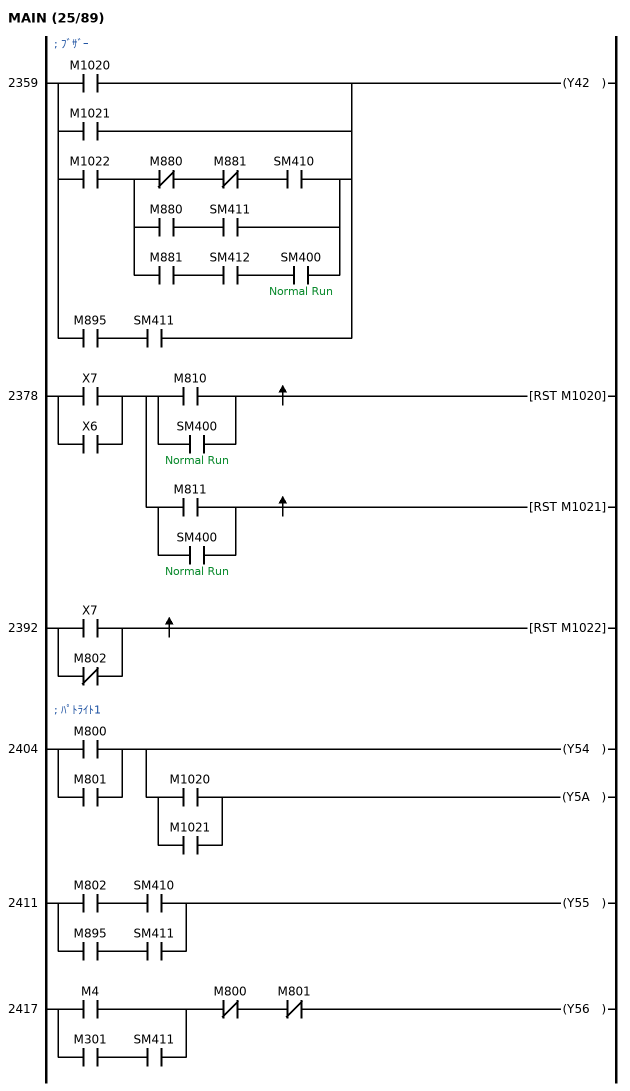
[picture p24: ladder of MAIN, rungs at steps 2359 to 2417]
; ﾌﾞｻﾞｰ
2359  LD      M1020
      OR      M1021
      LD      M1022
      LDI     M880
      ANI     M881
      AND     SM410
      LD      M880
      AND     SM411
      ORB
      LD      M881
      AND     SM412
      AND     SM400  ; Normal Run
      ORB
      ANB
      ORB
      LD      M895
      AND     SM411
      ORB
      OUT     Y42
2378  LD      X7
      OR      X6
      MPS
      LD      M810
      OR      SM400  ; Normal Run
      ANB
      MEP
      RST     M1020
      MPP
      LD      M811
      OR      SM400  ; Normal Run
      ANB
      MEP
      RST     M1021
2392  LD      X7
      ORI     M802
      MEP
      RST     M1022
; ﾊﾟﾄﾗｲﾄ1
2404  LD      M800
      OR      M801
      OUT     Y54
      LD      M1020
      OR      M1021
      ANB
      OUT     Y5A
2411  LD      M802
      AND     SM410
      LD      M895
      AND     SM411
      ORB
      OUT     Y55
2417  LD      M4
      LD      M301
      AND     SM411
      ORB
      ANI     M800
      ANI     M801
      OUT     Y56
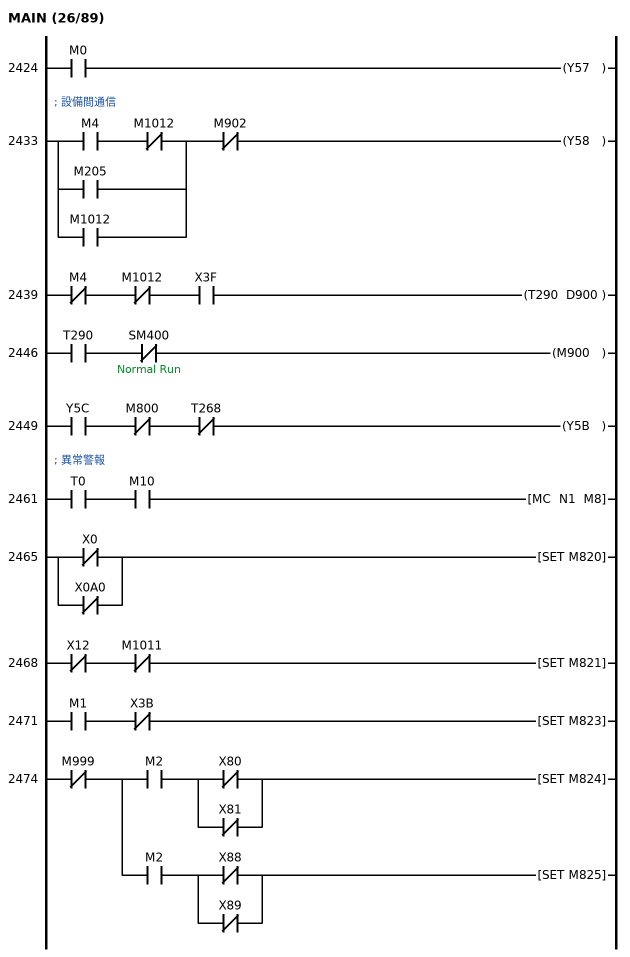
2424  LD      M0
      OUT     Y57
; 設備間通信
2433  LD      M4
      ANI     M1012
      OR      M205
      OR      M1012
      ANI     M902
      OUT     Y58
2439  LDI     M4
      ANI     M1012
      AND     X3F
      OUT     T290 D900
2446  LD      T290
      ANI     SM400  ; Normal Run
      OUT     M900
2449  LD      Y5C
      ANI     M800
      ANI     T268
      OUT     Y5B
; 異常警報
; 
2461  LD      T0
      AND     M10
      MC      N1 M8
2465  LDI     X0
      ORI     X0A0
      SET     M820
2468  LDI     X12
      ANI     M1011
      SET     M821
2471  LD      M1
      ANI     X3B
      SET     M823
2474  LDI     M999
      MPS
      AND     M2
      LDI     X80
      ORI     X81
      ANB
      SET     M824
      MPP
      AND     M2
      LDI     X88
      ORI     X89
      ANB
      SET     M825
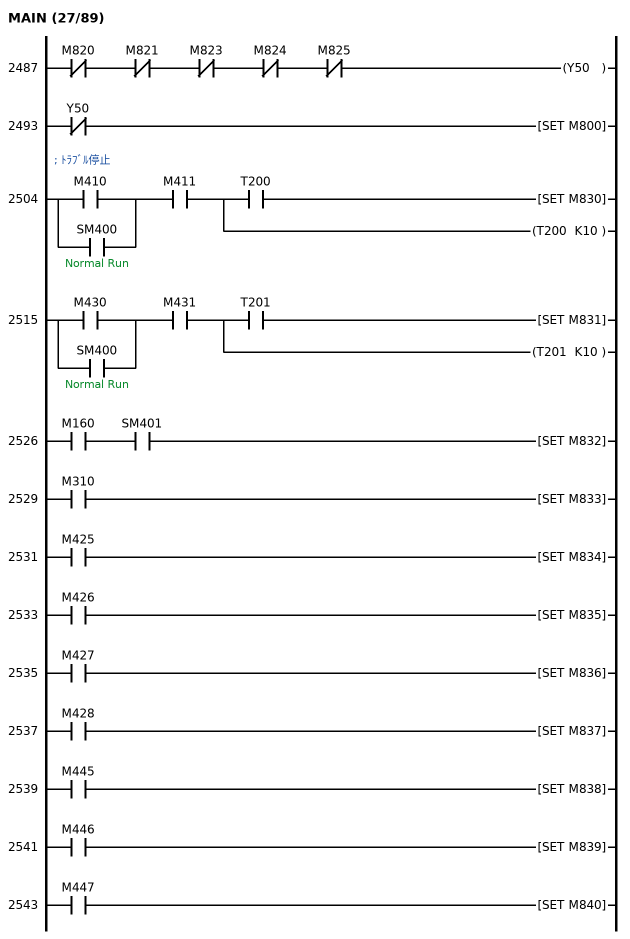
2487  LDI     M820
      ANI     M821
      ANI     M823
      ANI     M824
      ANI     M825
      OUT     Y50
2493  LDI     Y50
      SET     M800
; ﾄﾗﾌﾞﾙ停止
2504  LD      M410
      OR      SM400  ; Normal Run
      AND     M411
      MPS
      AND     T200
      SET     M830
      MPP
      OUT     T200 K10
2515  LD      M430
      OR      SM400  ; Normal Run
      AND     M431
      MPS
      AND     T201
      SET     M831
      MPP
      OUT     T201 K10
2526  LD      M160
      AND     SM401
      SET     M832
2529  LD      M310
      SET     M833
2531  LD      M425
      SET     M834
2533  LD      M426
      SET     M835
2535  LD      M427
      SET     M836
2537  LD      M428
      SET     M837
2539  LD      M445
      SET     M838
2541  LD      M446
      SET     M839
2543  LD      M447
      SET     M840
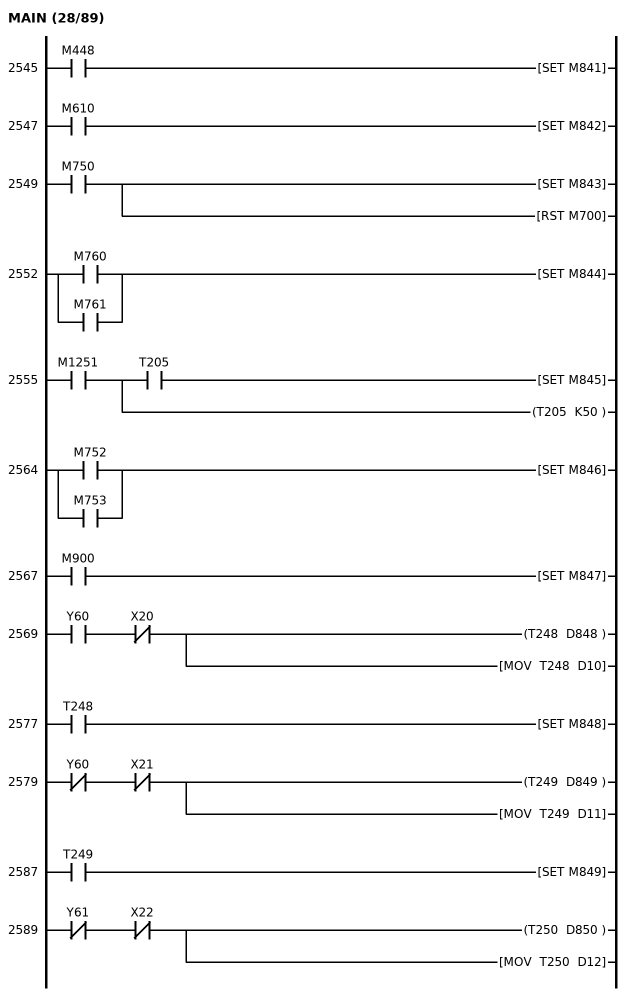
2545  LD      M448
      SET     M841
2547  LD      M610
      SET     M842
2549  LD      M750
      SET     M843
      RST     M700
2552  LD      M760
      OR      M761
      SET     M844
2555  LD      M1251
      MPS
      AND     T205
      SET     M845
      MPP
      OUT     T205 K50
2564  LD      M752
      OR      M753
      SET     M846
2567  LD      M900
      SET     M847
2569  LD      Y60
      ANI     X20
      OUT     T248 D848
      MOV     T248 D10
2577  LD      T248
      SET     M848
2579  LDI     Y60
      ANI     X21
      OUT     T249 D849
      MOV     T249 D11
2587  LD      T249
      SET     M849
2589  LDI     Y61
      ANI     X22
      OUT     T250 D850
      MOV     T250 D12
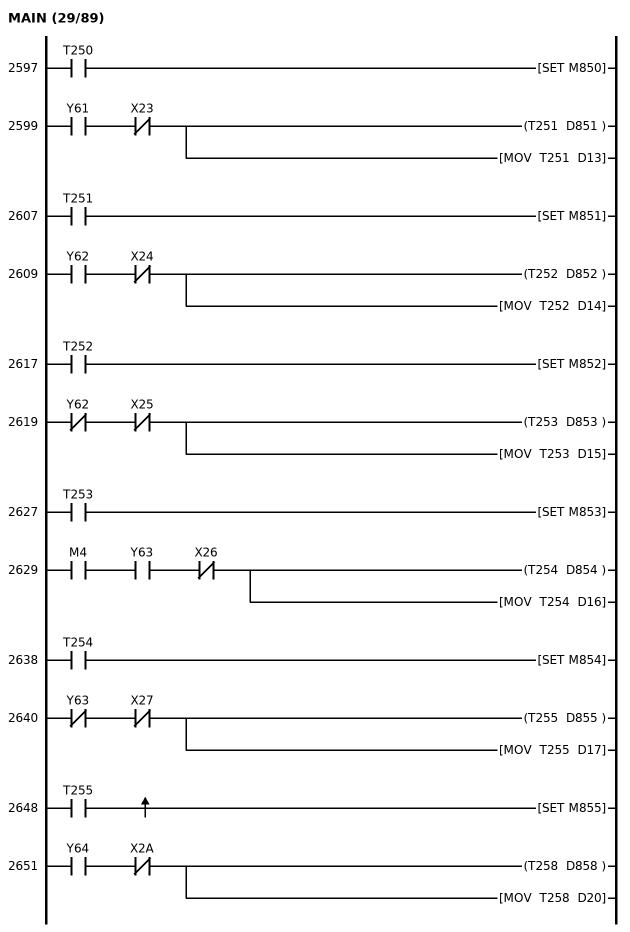
2597  LD      T250
      SET     M850
2599  LD      Y61
      ANI     X23
      OUT     T251 D851
      MOV     T251 D13
2607  LD      T251
      SET     M851
2609  LD      Y62
      ANI     X24
      OUT     T252 D852
      MOV     T252 D14
2617  LD      T252
      SET     M852
2619  LDI     Y62
      ANI     X25
      OUT     T253 D853
      MOV     T253 D15
2627  LD      T253
      SET     M853
2629  LD      M4
      AND     Y63
      ANI     X26
      OUT     T254 D854
      MOV     T254 D16
2638  LD      T254
      SET     M854
2640  LDI     Y63
      ANI     X27
      OUT     T255 D855
      MOV     T255 D17
2648  LD      T255
      MEP
      SET     M855
2651  LD      Y64
      ANI     X2A
      OUT     T258 D858
      MOV     T258 D20
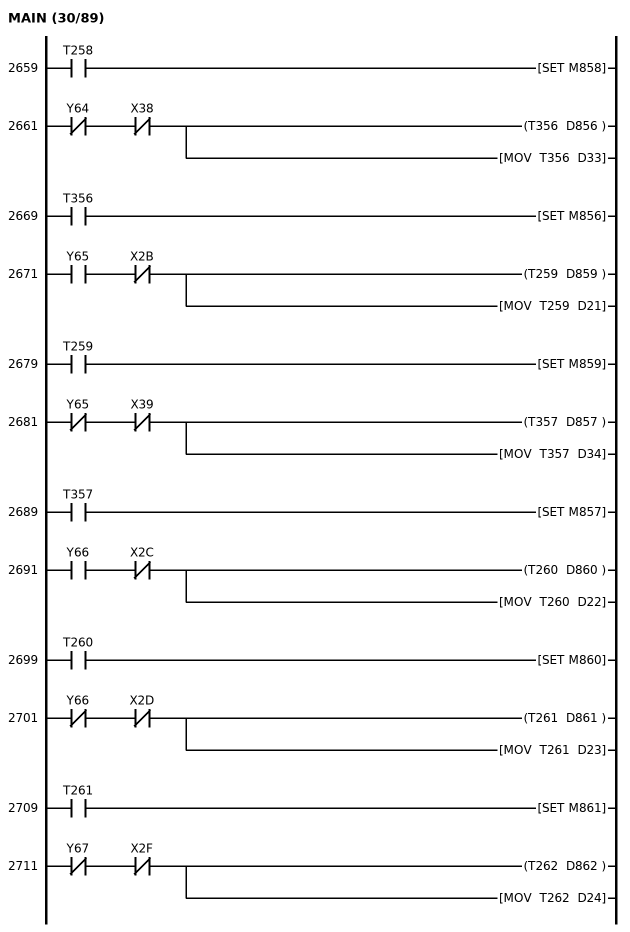
2659  LD      T258
      SET     M858
2661  LDI     Y64
      ANI     X38
      OUT     T356 D856
      MOV     T356 D33
2669  LD      T356
      SET     M856
2671  LD      Y65
      ANI     X2B
      OUT     T259 D859
      MOV     T259 D21
2679  LD      T259
      SET     M859
2681  LDI     Y65
      ANI     X39
      OUT     T357 D857
      MOV     T357 D34
2689  LD      T357
      SET     M857
2691  LD      Y66
      ANI     X2C
      OUT     T260 D860
      MOV     T260 D22
2699  LD      T260
      SET     M860
2701  LDI     Y66
      ANI     X2D
      OUT     T261 D861
      MOV     T261 D23
2709  LD      T261
      SET     M861
2711  LDI     Y67
      ANI     X2F
      OUT     T262 D862
      MOV     T262 D24
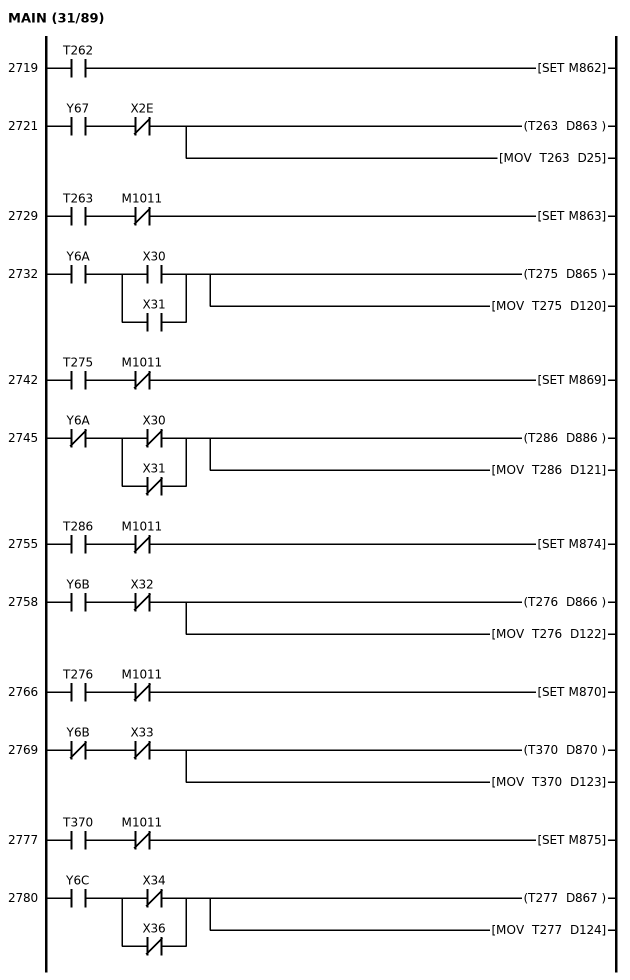
2719  LD      T262
      SET     M862
2721  LD      Y67
      ANI     X2E
      OUT     T263 D863
      MOV     T263 D25
2729  LD      T263
      ANI     M1011
      SET     M863
2732  LD      Y6A
      LD      X30
      OR      X31
      ANB
      OUT     T275 D865
      MOV     T275 D120
2742  LD      T275
      ANI     M1011
      SET     M869
2745  LDI     Y6A
      LDI     X30
      ORI     X31
      ANB
      OUT     T286 D886
      MOV     T286 D121
2755  LD      T286
      ANI     M1011
      SET     M874
2758  LD      Y6B
      ANI     X32
      OUT     T276 D866
      MOV     T276 D122
2766  LD      T276
      ANI     M1011
      SET     M870
2769  LDI     Y6B
      ANI     X33
      OUT     T370 D870
      MOV     T370 D123
2777  LD      T370
      ANI     M1011
      SET     M875
2780  LD      Y6C
      LDI     X34
      ORI     X36
      ANB
      OUT     T277 D867
      MOV     T277 D124
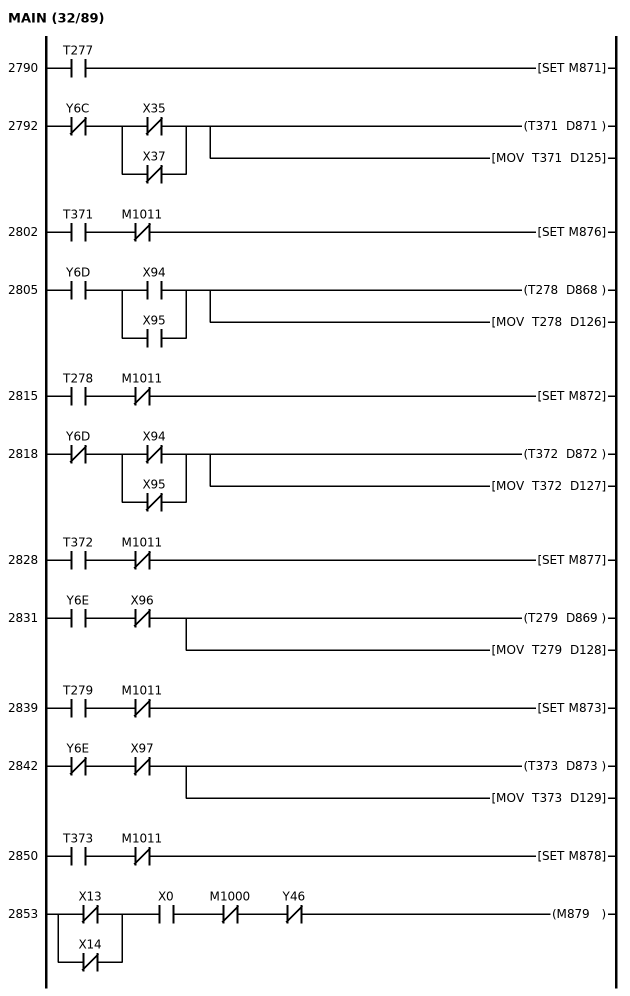
2790  LD      T277
      SET     M871
2792  LDI     Y6C
      LDI     X35
      ORI     X37
      ANB
      OUT     T371 D871
      MOV     T371 D125
2802  LD      T371
      ANI     M1011
      SET     M876
2805  LD      Y6D
      LD      X94
      OR      X95
      ANB
      OUT     T278 D868
      MOV     T278 D126
2815  LD      T278
      ANI     M1011
      SET     M872
2818  LDI     Y6D
      LDI     X94
      ORI     X95
      ANB
      OUT     T372 D872
      MOV     T372 D127
2828  LD      T372
      ANI     M1011
      SET     M877
2831  LD      Y6E
      ANI     X96
      OUT     T279 D869
      MOV     T279 D128
2839  LD      T279
      ANI     M1011
      SET     M873
2842  LDI     Y6E
      ANI     X97
      OUT     T373 D873
      MOV     T373 D129
2850  LD      T373
      ANI     M1011
      SET     M878
2853  LDI     X13
      ORI     X14
      AND     X0
      ANI     M1000
      ANI     Y46
      OUT     M879
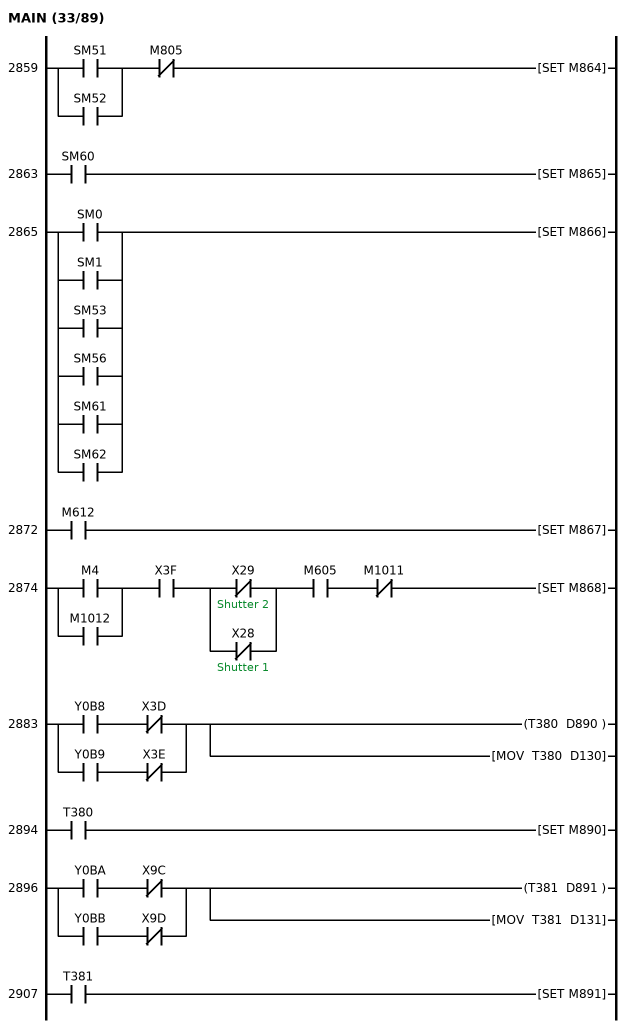
2859  LD      SM51
      OR      SM52
      ANI     M805
      SET     M864
2863  LD      SM60
      SET     M865
2865  LD      SM0
      OR      SM1
      OR      SM53
      OR      SM56
      OR      SM61
      OR      SM62
      SET     M866
2872  LD      M612
      SET     M867
2874  LD      M4
      OR      M1012
      AND     X3F
      LDI     X29  ; Shutter 2
      ORI     X28  ; Shutter 1
      ANB
      AND     M605
      ANI     M1011
      SET     M868
2883  LD      Y0B8
      ANI     X3D
      LD      Y0B9
      ANI     X3E
      ORB
      OUT     T380 D890
      MOV     T380 D130
2894  LD      T380
      SET     M890
2896  LD      Y0BA
      ANI     X9C
      LD      Y0BB
      ANI     X9D
      ORB
      OUT     T381 D891
      MOV     T381 D131
2907  LD      T381
      SET     M891
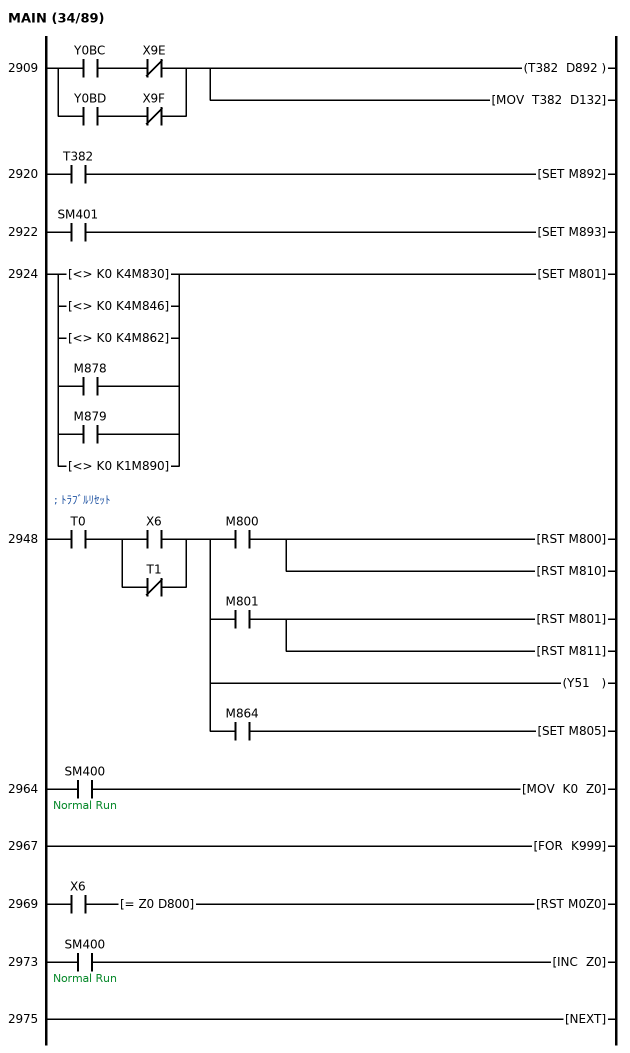
2909  LD      Y0BC
      ANI     X9E
      LD      Y0BD
      ANI     X9F
      ORB
      OUT     T382 D892
      MOV     T382 D132
2920  LD      T382
      SET     M892
2922  LD      SM401
      SET     M893
2924  LD<>    K0 K4M830
      OR<>    K0 K4M846
      OR<>    K0 K4M862
      OR      M878
      OR      M879
      OR<>    K0 K1M890
      SET     M801
; ﾄﾗﾌﾞﾙﾘｾｯﾄ
2948  LD      T0
      LD      X6
      ORI     T1
      ANB
      MPS
      AND     M800
      RST     M800
      RST     M810
      MRD
      AND     M801
      RST     M801
      RST     M811
      MPP
      OUT     Y51
      AND     M864
      SET     M805
2964  LD      SM400  ; Normal Run
      MOV     K0 Z0
2967  FOR     K999
2969  LD      X6
      AND=    Z0 D800
      RST     M0Z0
2973  LD      SM400  ; Normal Run
      INC     Z0
2975  NEXT
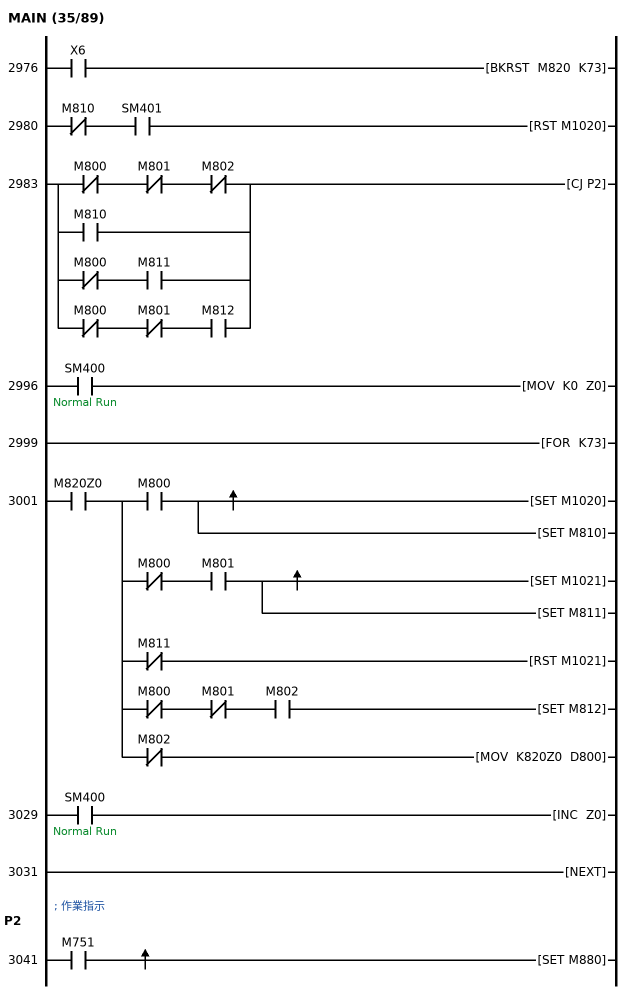
2976  LD      X6
      BKRST   M820 K73
2980  LDI     M810
      AND     SM401
      RST     M1020
2983  LDI     M800
      ANI     M801
      ANI     M802
      OR      M810
      LDI     M800
      AND     M811
      ORB
      LDI     M800
      ANI     M801
      AND     M812
      ORB
      CJ      P2
2996  LD      SM400  ; Normal Run
      MOV     K0 Z0
2999  FOR     K73
3001  LD      M820Z0
      MPS
      AND     M800
      MPS
      MEP
      SET     M1020
      MPP
      SET     M810
      MRD
      ANI     M800
      AND     M801
      MPS
      MEP
      SET     M1021
      MPP
      SET     M811
      MRD
      ANI     M811
      RST     M1021
      MRD
      ANI     M800
      ANI     M801
      AND     M802
      SET     M812
      MPP
      ANI     M802
      MOV     K820Z0 D800
3029  LD      SM400  ; Normal Run
      INC     Z0
3031  NEXT
      P2
; 作業指示
3041  LD      M751
      MEP
      SET     M880
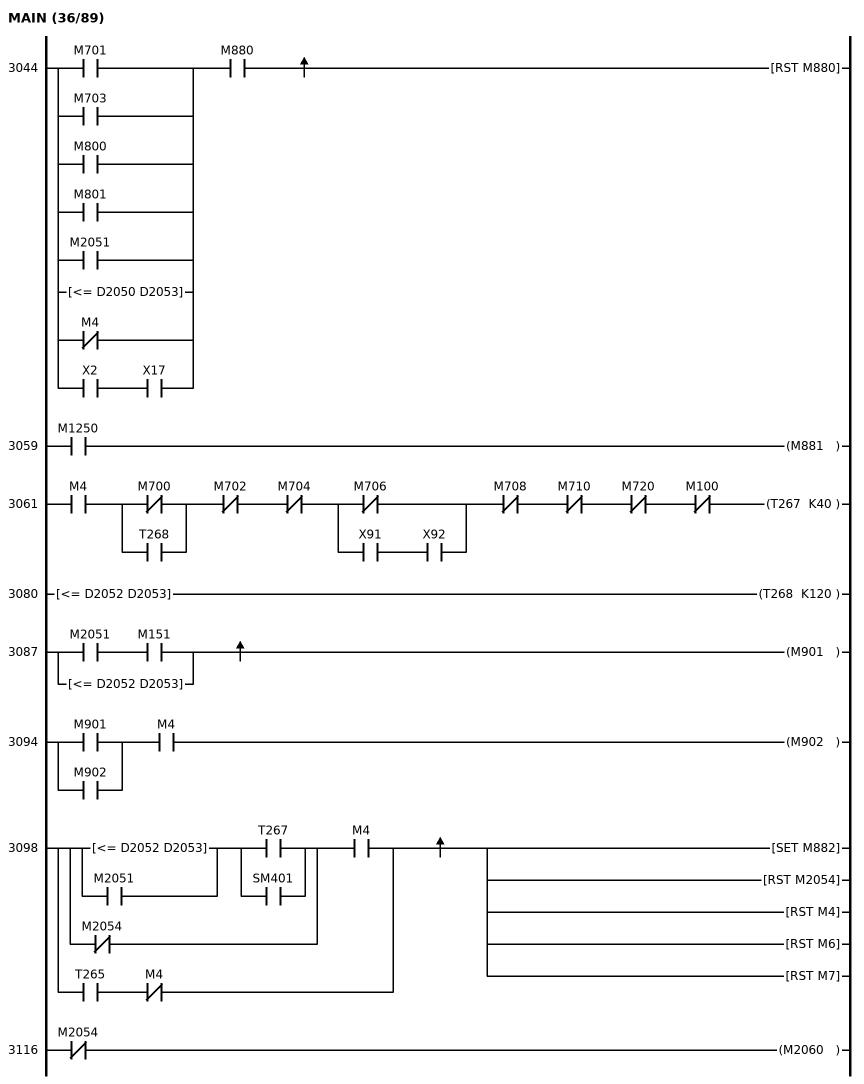
3044  LD      M701
      OR      M703
      OR      M800
      OR      M801
      OR      M2051
      OR<=    D2050 D2053
      ORI     M4
      LD      X2
      AND     X17
      ORB
      AND     M880
      MEP
      RST     M880
3059  LD      M1250
      OUT     M881
3061  LD      M4
      LDI     M700
      OR      T268
      ANB
      ANI     M702
      ANI     M704
      LDI     M706
      LD      X91
      AND     X92
      ORB
      ANB
      ANI     M708
      ANI     M710
      ANI     M720
      ANI     M100
      OUT     T267 K40
3080  LD<=    D2052 D2053
      OUT     T268 K120
3087  LD      M2051
      AND     M151
      OR<=    D2052 D2053
      MEP
      OUT     M901
3094  LD      M901
      OR      M902
      AND     M4
      OUT     M902
3098  LD<=    D2052 D2053
      OR      M2051
      LD      T267
      OR      SM401
      ANB
      ORI     M2054
      AND     M4
      LD      T265
      ANI     M4
      ORB
      MEP
      SET     M882
      RST     M2054
      RST     M4
      RST     M6
      RST     M7
3116  LDI     M2054
      OUT     M2060
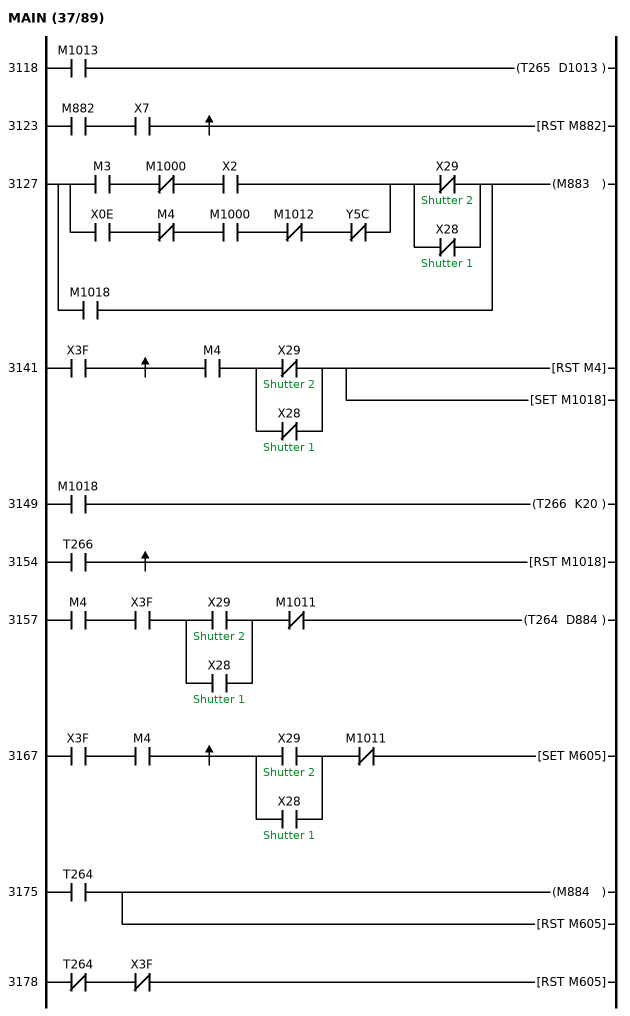
3118  LD      M1013
      OUT     T265 D1013
3123  LD      M882
      AND     X7
      MEP
      RST     M882
3127  LD      M3
      ANI     M1000
      AND     X2
      LD      X0E
      ANI     M4
      AND     M1000
      ANI     M1012
      ANI     Y5C
      ORB
      LDI     X29  ; Shutter 2
      ORI     X28  ; Shutter 1
      ANB
      OR      M1018
      OUT     M883
3141  LD      X3F
      MEP
      AND     M4
      LDI     X29  ; Shutter 2
      ORI     X28  ; Shutter 1
      ANB
      RST     M4
      SET     M1018
3149  LD      M1018
      OUT     T266 K20
3154  LD      T266
      MEP
      RST     M1018
3157  LD      M4
      AND     X3F
      LD      X29  ; Shutter 2
      OR      X28  ; Shutter 1
      ANB
      ANI     M1011
      OUT     T264 D884
3167  LD      X3F
      AND     M4
      MEP
      LD      X29  ; Shutter 2
      OR      X28  ; Shutter 1
      ANB
      ANI     M1011
      SET     M605
3175  LD      T264
      OUT     M884
      RST     M605
3178  LDI     T264
      ANI     X3F
      RST     M605
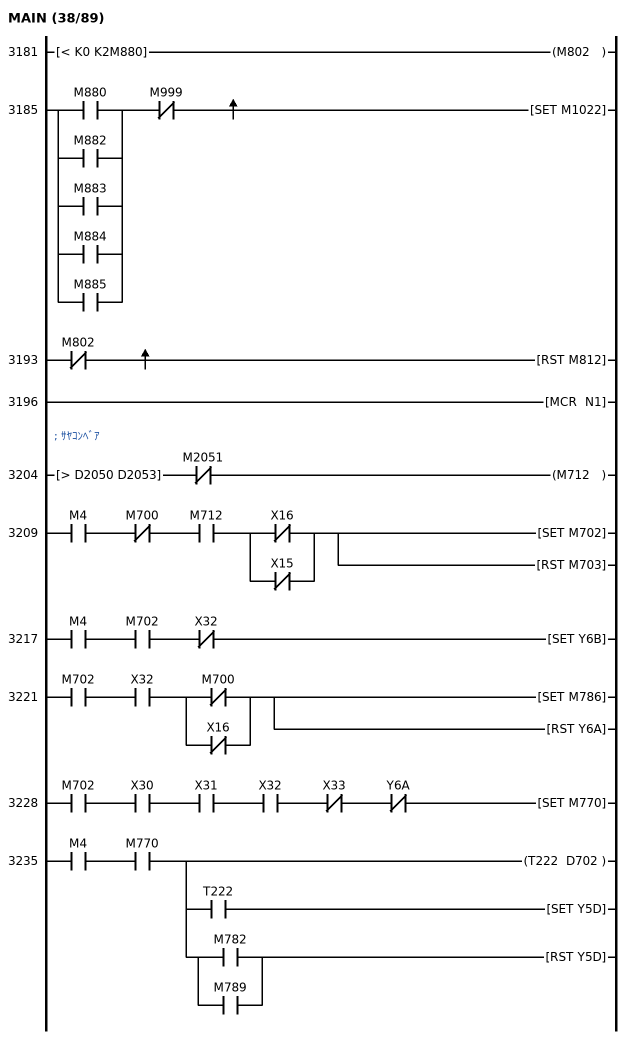
3181  LD<     K0 K2M880
      OUT     M802
3185  LD      M880
      OR      M882
      OR      M883
      OR      M884
      OR      M885
      ANI     M999
      MEP
      SET     M1022
3193  LDI     M802
      MEP
      RST     M812
3196  MCR     N1
; ｻﾔｺﾝﾍﾞｱ
; 
3204  LD>     D2050 D2053
      ANI     M2051
      OUT     M712
3209  LD      M4
      ANI     M700
      AND     M712
      LDI     X16
      ORI     X15
      ANB
      SET     M702
      RST     M703
3217  LD      M4
      AND     M702
      ANI     X32
      SET     Y6B
3221  LD      M702
      AND     X32
      LDI     M700
      ORI     X16
      ANB
      SET     M786
      RST     Y6A
3228  LD      M702
      AND     X30
      AND     X31
      AND     X32
      ANI     X33
      ANI     Y6A
      SET     M770
3235  LD      M4
      AND     M770
      OUT     T222 D702
      MPS
      AND     T222
      SET     Y5D
      MPP
      LD      M782
      OR      M789
      ANB
      RST     Y5D
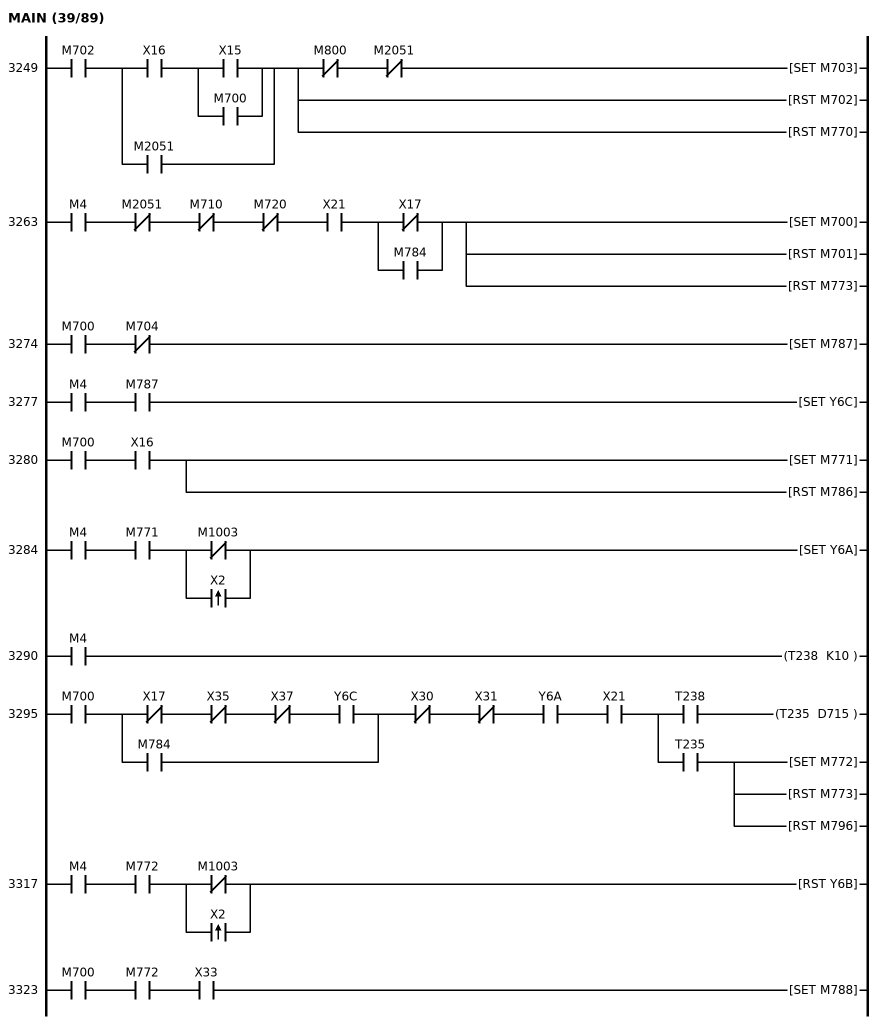
3249  LD      M702
      LD      X16
      LD      X15
      OR      M700
      ANB
      OR      M2051
      ANB
      MPS
      ANI     M800
      ANI     M2051
      SET     M703
      MPP
      RST     M702
      RST     M770
3263  LD      M4
      ANI     M2051
      ANI     M710
      ANI     M720
      AND     X21
      LDI     X17
      OR      M784
      ANB
      SET     M700
      RST     M701
      RST     M773
3274  LD      M700
      ANI     M704
      SET     M787
3277  LD      M4
      AND     M787
      SET     Y6C
3280  LD      M700
      AND     X16
      SET     M771
      RST     M786
3284  LD      M4
      AND     M771
      LDI     M1003
      ORP     X2
      ANB
      SET     Y6A
3290  LD      M4
      OUT     T238 K10
3295  LD      M700
      LDI     X17
      ANI     X35
      ANI     X37
      AND     Y6C
      OR      M784
      ANB
      ANI     X30
      ANI     X31
      AND     Y6A
      AND     X21
      MPS
      AND     T238
      OUT     T235 D715
      MPP
      AND     T235
      SET     M772
      RST     M773
      RST     M796
3317  LD      M4
      AND     M772
      LDI     M1003
      ORP     X2
      ANB
      RST     Y6B
3323  LD      M700
      AND     M772
      AND     X33
      SET     M788
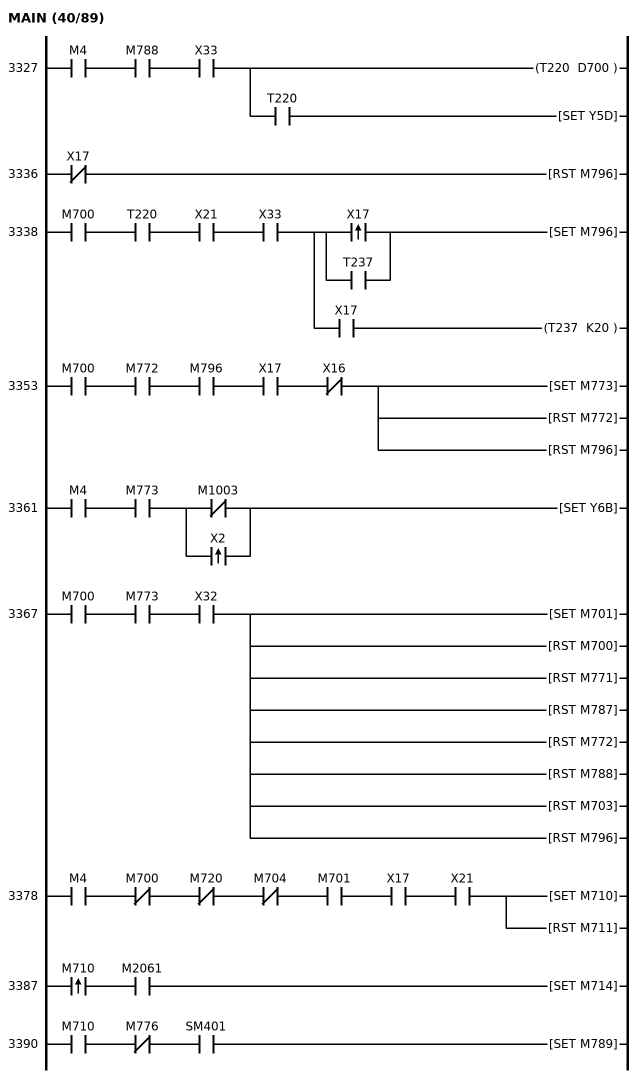
3327  LD      M4
      AND     M788
      AND     X33
      OUT     T220 D700
      AND     T220
      SET     Y5D
3336  LDI     X17
      RST     M796
3338  LD      M700
      AND     T220
      AND     X21
      AND     X33
      MPS
      LDP     X17
      OR      T237
      ANB
      SET     M796
      MPP
      AND     X17
      OUT     T237 K20
3353  LD      M700
      AND     M772
      AND     M796
      AND     X17
      ANI     X16
      SET     M773
      RST     M772
      RST     M796
3361  LD      M4
      AND     M773
      LDI     M1003
      ORP     X2
      ANB
      SET     Y6B
3367  LD      M700
      AND     M773
      AND     X32
      SET     M701
      RST     M700
      RST     M771
      RST     M787
      RST     M772
      RST     M788
      RST     M703
      RST     M796
3378  LD      M4
      ANI     M700
      ANI     M720
      ANI     M704
      AND     M701
      AND     X17
      AND     X21
      SET     M710
      RST     M711
3387  LDP     M710
      AND     M2061
      SET     M714
3390  LD      M710
      ANI     M776
      AND     SM401
      SET     M789
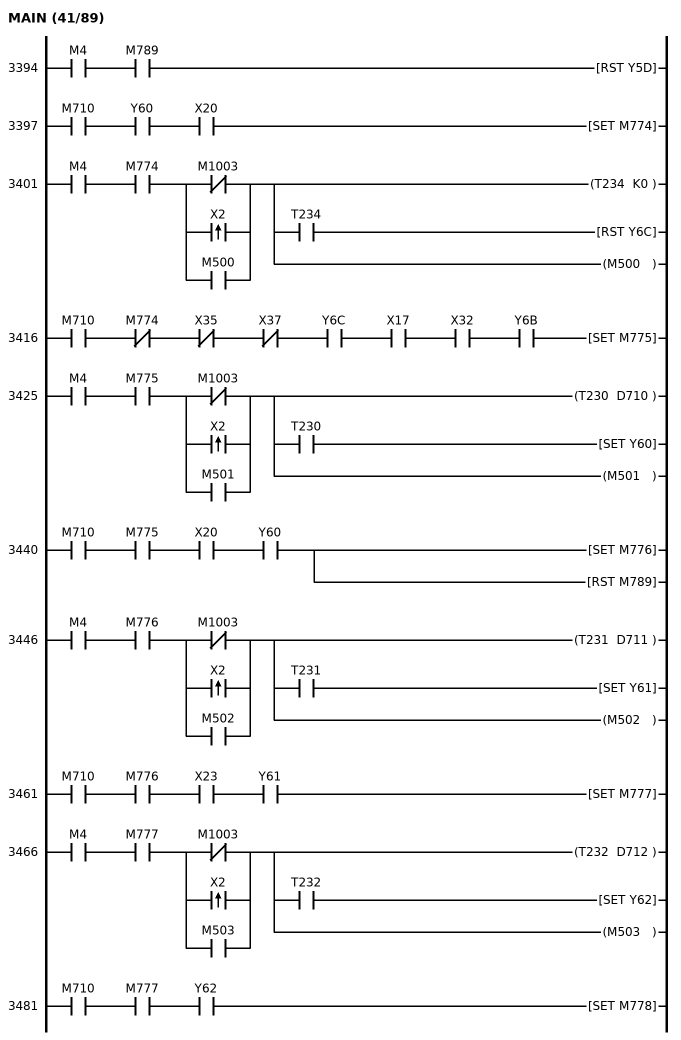
3394  LD      M4
      AND     M789
      RST     Y5D
3397  LD      M710
      AND     Y60
      AND     X20
      SET     M774
3401  LD      M4
      AND     M774
      LDI     M1003
      ORP     X2
      OR      M500
      ANB
      OUT     T234 K0
      MPS
      AND     T234
      RST     Y6C
      MPP
      OUT     M500
3416  LD      M710
      ANI     M774
      ANI     X35
      ANI     X37
      AND     Y6C
      AND     X17
      AND     X32
      AND     Y6B
      SET     M775
3425  LD      M4
      AND     M775
      LDI     M1003
      ORP     X2
      OR      M501
      ANB
      OUT     T230 D710
      MPS
      AND     T230
      SET     Y60
      MPP
      OUT     M501
3440  LD      M710
      AND     M775
      AND     X20
      AND     Y60
      SET     M776
      RST     M789
3446  LD      M4
      AND     M776
      LDI     M1003
      ORP     X2
      OR      M502
      ANB
      OUT     T231 D711
      MPS
      AND     T231
      SET     Y61
      MPP
      OUT     M502
3461  LD      M710
      AND     M776
      AND     X23
      AND     Y61
      SET     M777
3466  LD      M4
      AND     M777
      LDI     M1003
      ORP     X2
      OR      M503
      ANB
      OUT     T232 D712
      MPS
      AND     T232
      SET     Y62
      MPP
      OUT     M503
3481  LD      M710
      AND     M777
      AND     Y62
      SET     M778
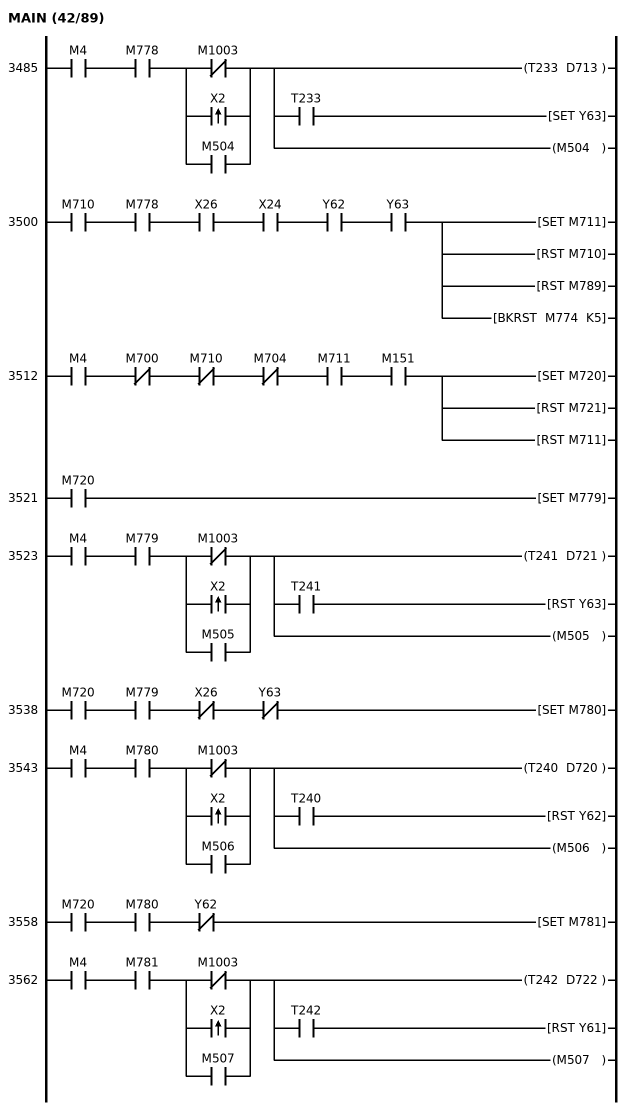
3485  LD      M4
      AND     M778
      LDI     M1003
      ORP     X2
      OR      M504
      ANB
      OUT     T233 D713
      MPS
      AND     T233
      SET     Y63
      MPP
      OUT     M504
3500  LD      M710
      AND     M778
      AND     X26
      AND     X24
      AND     Y62
      AND     Y63
      SET     M711
      RST     M710
      RST     M789
      BKRST   M774 K5
3512  LD      M4
      ANI     M700
      ANI     M710
      ANI     M704
      AND     M711
      AND     M151
      SET     M720
      RST     M721
      RST     M711
3521  LD      M720
      SET     M779
3523  LD      M4
      AND     M779
      LDI     M1003
      ORP     X2
      OR      M505
      ANB
      OUT     T241 D721
      MPS
      AND     T241
      RST     Y63
      MPP
      OUT     M505
3538  LD      M720
      AND     M779
      ANI     X26
      ANI     Y63
      SET     M780
3543  LD      M4
      AND     M780
      LDI     M1003
      ORP     X2
      OR      M506
      ANB
      OUT     T240 D720
      MPS
      AND     T240
      RST     Y62
      MPP
      OUT     M506
3558  LD      M720
      AND     M780
      ANI     Y62
      SET     M781
3562  LD      M4
      AND     M781
      LDI     M1003
      ORP     X2
      OR      M507
      ANB
      OUT     T242 D722
      MPS
      AND     T242
      RST     Y61
      MPP
      OUT     M507
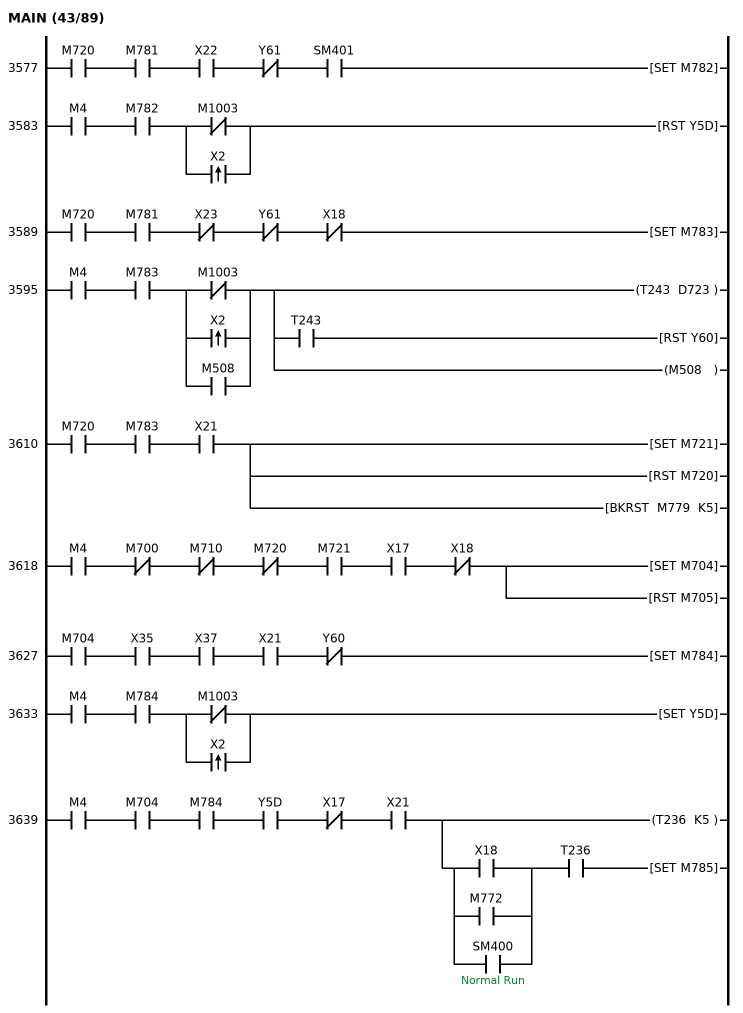
3577  LD      M720
      AND     M781
      AND     X22
      ANI     Y61
      AND     SM401
      SET     M782
3583  LD      M4
      AND     M782
      LDI     M1003
      ORP     X2
      ANB
      RST     Y5D
3589  LD      M720
      AND     M781
      ANI     X23
      ANI     Y61
      ANI     X18
      SET     M783
3595  LD      M4
      AND     M783
      LDI     M1003
      ORP     X2
      OR      M508
      ANB
      OUT     T243 D723
      MPS
      AND     T243
      RST     Y60
      MPP
      OUT     M508
3610  LD      M720
      AND     M783
      AND     X21
      SET     M721
      RST     M720
      BKRST   M779 K5
3618  LD      M4
      ANI     M700
      ANI     M710
      ANI     M720
      AND     M721
      AND     X17
      ANI     X18
      SET     M704
      RST     M705
3627  LD      M704
      AND     X35
      AND     X37
      AND     X21
      ANI     Y60
      SET     M784
3633  LD      M4
      AND     M784
      LDI     M1003
      ORP     X2
      ANB
      SET     Y5D
3639  LD      M4
      AND     M704
      AND     M784
      AND     Y5D
      ANI     X17
      AND     X21
      OUT     T236 K5
      LD      X18
      OR      M772
      OR      SM400  ; Normal Run
      ANB
      AND     T236
      SET     M785
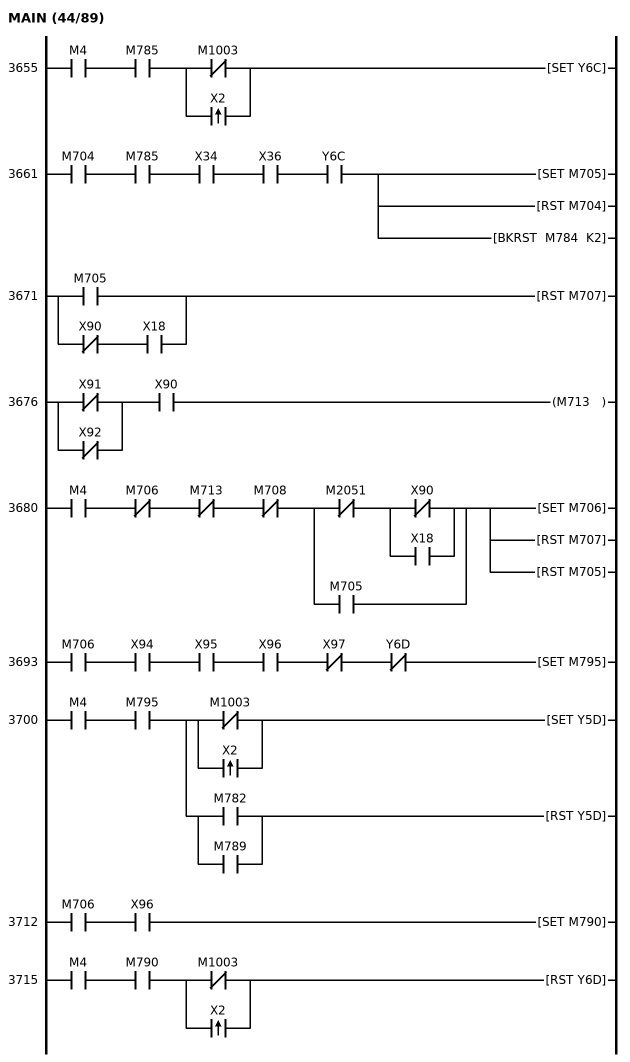
3655  LD      M4
      AND     M785
      LDI     M1003
      ORP     X2
      ANB
      SET     Y6C
3661  LD      M704
      AND     M785
      AND     X34
      AND     X36
      AND     Y6C
      SET     M705
      RST     M704
      BKRST   M784 K2
3671  LD      M705
      LDI     X90
      AND     X18
      ORB
      RST     M707
3676  LDI     X91
      ORI     X92
      AND     X90
      OUT     M713
3680  LD      M4
      ANI     M706
      ANI     M713
      ANI     M708
      LDI     M2051
      LDI     X90
      OR      X18
      ANB
      OR      M705
      ANB
      SET     M706
      RST     M707
      RST     M705
3693  LD      M706
      AND     X94
      AND     X95
      AND     X96
      ANI     X97
      ANI     Y6D
      SET     M795
3700  LD      M4
      AND     M795
      MPS
      LDI     M1003
      ORP     X2
      ANB
      SET     Y5D
      MPP
      LD      M782
      OR      M789
      ANB
      RST     Y5D
3712  LD      M706
      AND     X96
      SET     M790
3715  LD      M4
      AND     M790
      LDI     M1003
      ORP     X2
      ANB
      RST     Y6D
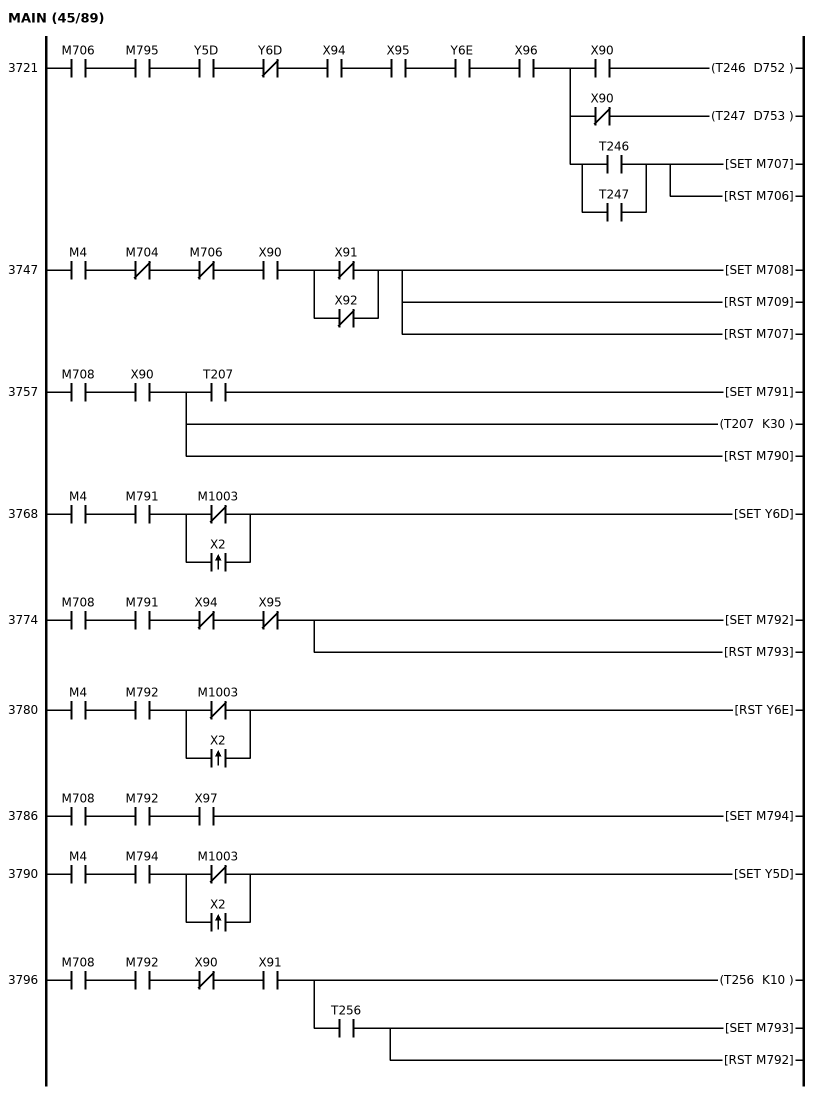
3721  LD      M706
      AND     M795
      AND     Y5D
      ANI     Y6D
      AND     X94
      AND     X95
      AND     Y6E
      AND     X96
      MPS
      AND     X90
      OUT     T246 D752
      MRD
      ANI     X90
      OUT     T247 D753
      MPP
      LD      T246
      OR      T247
      ANB
      SET     M707
      RST     M706
3747  LD      M4
      ANI     M704
      ANI     M706
      AND     X90
      LDI     X91
      ORI     X92
      ANB
      SET     M708
      RST     M709
      RST     M707
3757  LD      M708
      AND     X90
      MPS
      AND     T207
      SET     M791
      MPP
      OUT     T207 K30
      RST     M790
3768  LD      M4
      AND     M791
      LDI     M1003
      ORP     X2
      ANB
      SET     Y6D
3774  LD      M708
      AND     M791
      ANI     X94
      ANI     X95
      SET     M792
      RST     M793
3780  LD      M4
      AND     M792
      LDI     M1003
      ORP     X2
      ANB
      RST     Y6E
3786  LD      M708
      AND     M792
      AND     X97
      SET     M794
3790  LD      M4
      AND     M794
      LDI     M1003
      ORP     X2
      ANB
      SET     Y5D
3796  LD      M708
      AND     M792
      ANI     X90
      AND     X91
      OUT     T256 K10
      AND     T256
      SET     M793
      RST     M792
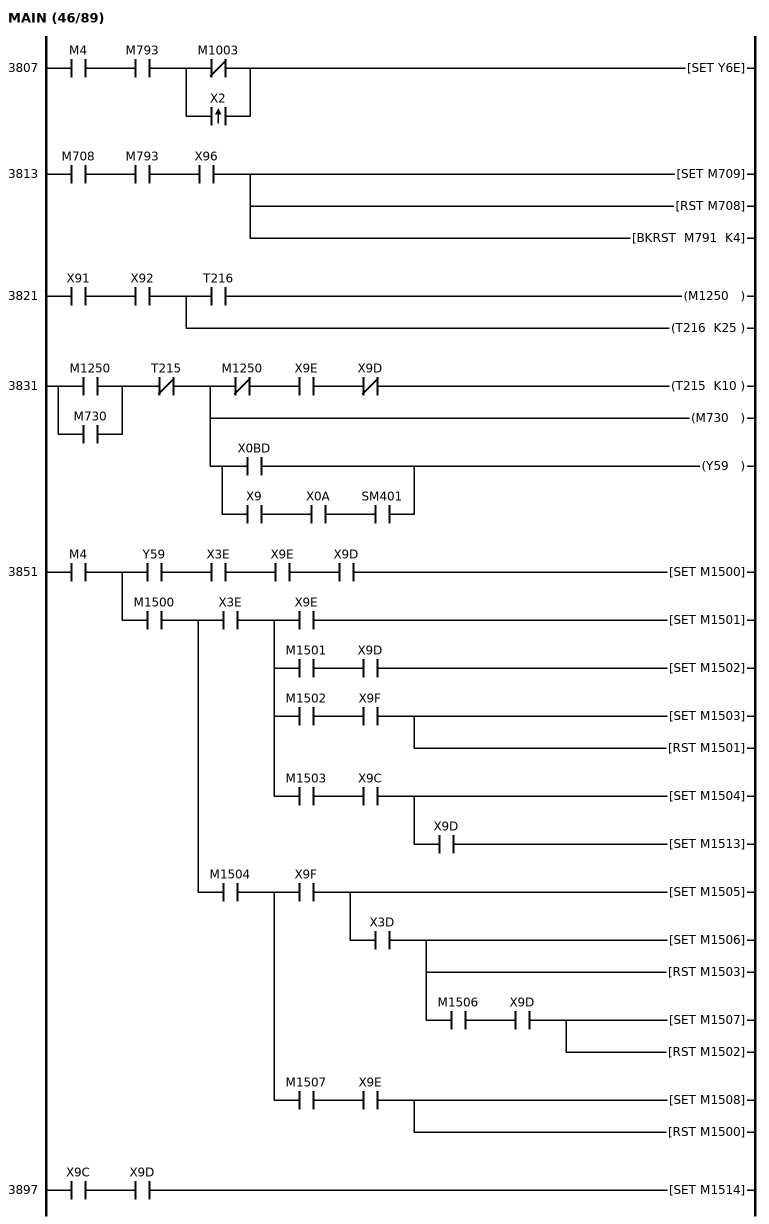
3807  LD      M4
      AND     M793
      LDI     M1003
      ORP     X2
      ANB
      SET     Y6E
3813  LD      M708
      AND     M793
      AND     X96
      SET     M709
      RST     M708
      BKRST   M791 K4
3821  LD      X91
      AND     X92
      MPS
      AND     T216
      OUT     M1250
      MPP
      OUT     T216 K25
3831  LD      M1250
      OR      M730
      ANI     T215
      MPS
      ANI     M1250
      AND     X9E
      ANI     X9D
      OUT     T215 K10
      MPP
      OUT     M730
      LD      X0BD
      LD      X9
      AND     X0A
      AND     SM401
      ORB
      ANB
      OUT     Y59
3851  LD      M4
      MPS
      AND     Y59
      AND     X3E
      AND     X9E
      AND     X9D
      SET     M1500
      MPP
      AND     M1500
      MPS
      AND     X3E
      MPS
      AND     X9E
      SET     M1501
      MRD
      AND     M1501
      AND     X9D
      SET     M1502
      MRD
      AND     M1502
      AND     X9F
      SET     M1503
      RST     M1501
      MPP
      AND     M1503
      AND     X9C
      SET     M1504
      AND     X9D
      SET     M1513
      MPP
      AND     M1504
      MPS
      AND     X9F
      SET     M1505
      AND     X3D
      SET     M1506
      RST     M1503
      AND     M1506
      AND     X9D
      SET     M1507
      RST     M1502
      MPP
      AND     M1507
      AND     X9E
      SET     M1508
      RST     M1500
3897  LD      X9C
      AND     X9D
      SET     M1514
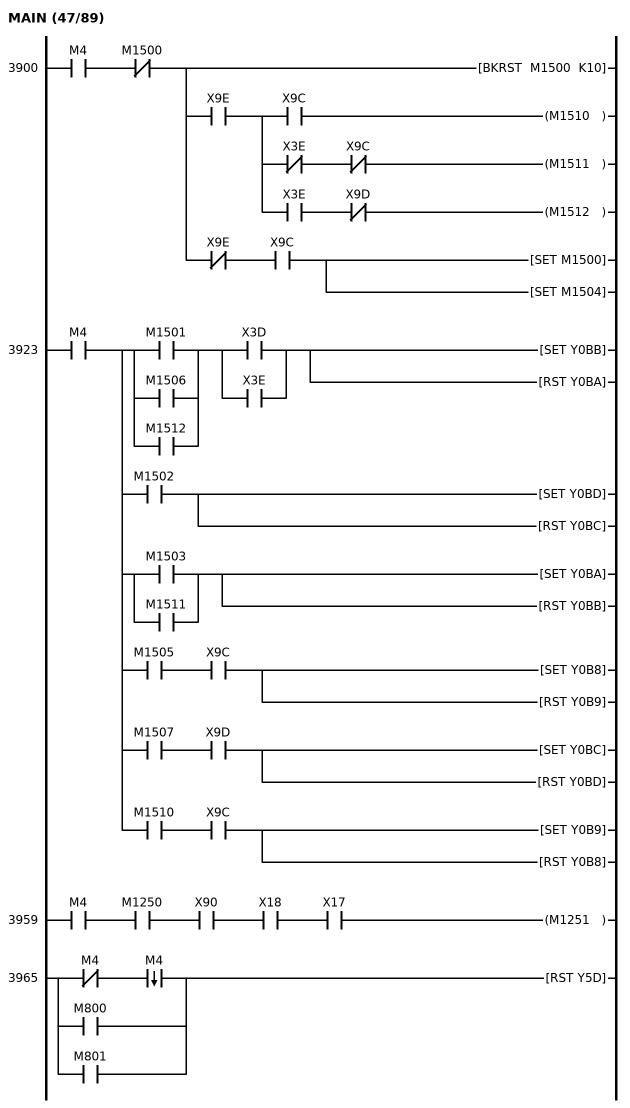
3900  LD      M4
      ANI     M1500
      BKRST   M1500 K10
      MPS
      AND     X9E
      MPS
      AND     X9C
      OUT     M1510
      MRD
      ANI     X3E
      ANI     X9C
      OUT     M1511
      MPP
      AND     X3E
      ANI     X9D
      OUT     M1512
      MPP
      ANI     X9E
      AND     X9C
      SET     M1500
      SET     M1504
3923  LD      M4
      MPS
      LD      M1501
      OR      M1506
      OR      M1512
      ANB
      LD      X3D
      OR      X3E
      ANB
      SET     Y0BB
      RST     Y0BA
      MRD
      AND     M1502
      SET     Y0BD
      RST     Y0BC
      MRD
      LD      M1503
      OR      M1511
      ANB
      SET     Y0BA
      RST     Y0BB
      MRD
      AND     M1505
      AND     X9C
      SET     Y0B8
      RST     Y0B9
      MRD
      AND     M1507
      AND     X9D
      SET     Y0BC
      RST     Y0BD
      MPP
      AND     M1510
      AND     X9C
      SET     Y0B9
      RST     Y0B8
3959  LD      M4
      AND     M1250
      AND     X90
      AND     X18
      AND     X17
      OUT     M1251
3965  LDI     M4
      ANDF    M4
      OR      M800
      OR      M801
      RST     Y5D
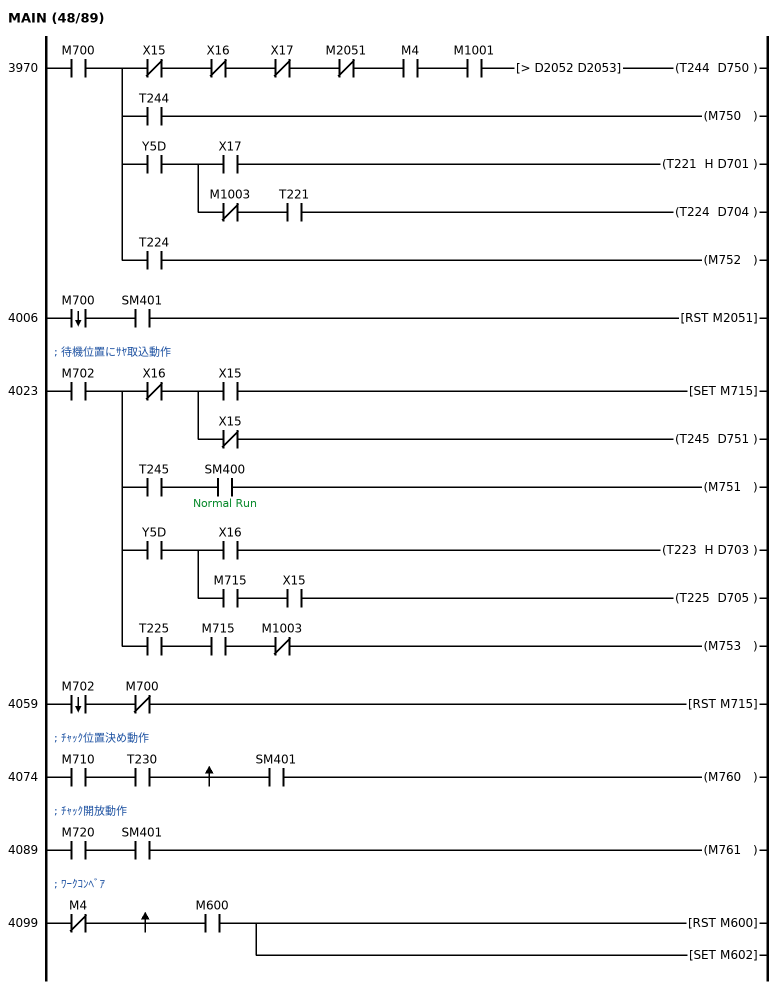
3970  LD      M700
      MPS
      ANI     X15
      ANI     X16
      ANI     X17
      ANI     M2051
      AND     M4
      AND     M1001
      AND>    D2052 D2053
      OUT     T244 D750
      MRD
      AND     T244
      OUT     M750
      MRD
      AND     Y5D
      MPS
      AND     X17
      OUTH    T221 D701
      MPP
      ANI     M1003
      AND     T221
      OUT     T224 D704
      MPP
      AND     T224
      OUT     M752
4006  LDF     M700
      AND     SM401
      RST     M2051
; 待機位置にｻﾔ取込動作
4023  LD      M702
      MPS
      ANI     X16
      MPS
      AND     X15
      SET     M715
      MPP
      ANI     X15
      OUT     T245 D751
      MRD
      AND     T245
      AND     SM400  ; Normal Run
      OUT     M751
      MRD
      AND     Y5D
      MPS
      AND     X16
      OUTH    T223 D703
      MPP
      AND     M715
      AND     X15
      OUT     T225 D705
      MPP
      AND     T225
      AND     M715
      ANI     M1003
      OUT     M753
4059  LDF     M702
      ANI     M700
      RST     M715
; ﾁｬｯｸ位置決め動作
4074  LD      M710
      AND     T230
      MEP
      AND     SM401
      OUT     M760
; ﾁｬｯｸ開放動作
4089  LD      M720
      AND     SM401
      OUT     M761
; ﾜｰｸｺﾝﾍﾞｱ
; 
4099  LDI     M4
      MEP
      AND     M600
      RST     M600
      SET     M602
